PROGRAM MAIN
VAR
END_VAR

MainPlay();

END_PROGRAM

(* stored: Version 1.1.0.1
   POU MAIN: Id {cff1dec8-1ada-47de-8f2e-f328f293d9c3}, SpecialFunc None *)
